FUNCTION_BLOCK EK1200
VAR_INPUT
	En: BOOL;
END_VAR
VAR_OUTPUT
	EnO: BOOL;
END_VAR

EnO:=En;

END_FUNCTION_BLOCK

(* stored: Version 1.1.0.1, ProductVersion 3.1.4022.6
   POU EK1200: Id {98544b5d-cfdf-476a-90c0-230bdaff0ec8}, SpecialFunc None *)
